FUNCTION_BLOCK TcoCylinderMoveTask EXTENDS TcoCore.TcoTask
VAR_INPUT
    PositionSensor         : BOOL;
    MaxTimeToReachPosition : TIME := T#10S;
    TimeToRefill           : TIME := T#100MS;
    PositionName           : STRING(25);
END_VAR
VAR_IN_OUT
    MoveToPositionSignal : BOOL;
    InverseSignal        : BOOL;
END_VAR

VAR
    _stringBuilder : TcoCore.StringBuilder;
END_VAR

IF (THIS^.Execute()) THEN
    IF (THIS^.ElapsedTime > MaxTimeToReachPosition) THEN
        THIS^.Messenger
            .Warning(_stringBuilder.Clear().Append(PositionName).Append(' sensor not reached yet.').ToString());
    END_IF;

    InverseSignal        := FALSE;
    MoveToPositionSignal := TRUE;
    THIS^.DoneWhen(PositionSensor);
END_IF

METHOD PUBLIC FB_init : BOOL
VAR_INPUT
    bInitRetains : BOOL; // if TRUE, the retain variables are initialized (warm start / cold start)
    bInCopyCode  : BOOL; // if TRUE, the instance afterwards gets moved into the copy code (online change)
    ParentObject : ITcoObject;
END_VAR
END_METHOD

(*~
    <docu>
        <summary>
            Executes when task is aborted.
        </summary>
    </docu>
~*)
METHOD PROTECTED OnAbort
MoveToPositionSignal := FALSE;
END_METHOD

METHOD PROTECTED OnError
END_METHOD

METHOD PROTECTED OnStart
END_METHOD

END_FUNCTION_BLOCK

(* stored: Version 1.1.0.1, ProductVersion 3.1.4024.12
   POU TcoCylinderMoveTask: Id {01a071c3-2da6-46ad-bcae-667cb69126ec}, SpecialFunc None
   Method FB_init: Id {f807fc31-6cbf-4d2c-89b3-3f2e7f2cbe06}
   Method OnAbort: Id {72bfa40f-fbda-4149-a8ac-f5f4c6901e79}
   Method OnError: Id {f05a36ca-418b-4e3e-b167-beca7f629a5d}
   Method OnStart: Id {d0a840d1-4bf6-4b25-948d-c8823767156f} *)
